FUNCTION_BLOCK PnpCylinders (* Composite Function Block Type *)
  (* Standard: 61499-2 *)
  (* Version 0.0, 2/7/2012, XPMUser, nxtControl GmbH, template *)
  PACKAGE Main;
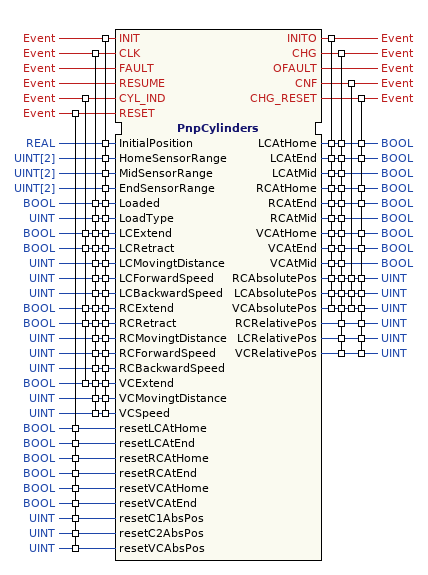
  EVENT_INPUT
    INIT WITH LCForwardSpeed, LCBackwardSpeed, LCExtend, LCRetract, LCMovingtDistance, HomeSensorRange, EndSensorRange, InitialPosition, LoadType, Loaded, MidSensorRange, RCForwardSpeed, RCBackwardSpeed, RCExtend, RCRetract, RCMovingtDistance, VCSpeed, VCExtend, VCMovingtDistance; (* Initialization Request *)
    CLK WITH Loaded, LoadType, LCExtend, LCRetract, LCMovingtDistance, LCForwardSpeed, LCBackwardSpeed, RCExtend, RCRetract, RCMovingtDistance, RCForwardSpeed, RCBackwardSpeed, VCExtend, VCMovingtDistance, VCSpeed;
    FAULT;
    RESUME;
    CYL_IND WITH LCExtend, LCRetract, RCExtend, RCRetract, VCExtend;
    RESET WITH resetLCAtHome, resetLCAtEnd, resetRCAtHome, resetRCAtEnd, resetVCAtHome, resetVCAtEnd, resetC1AbsPos, resetC2AbsPos, resetVCAbsPos;
  END_EVENT
  EVENT_OUTPUT
    INITO WITH LCAtHome, LCAtEnd, LCAtMid, RCAtHome, RCAtEnd, RCAtMid, VCAtHome, VCAtEnd, VCAtMid, RCAbsolutePos, LCAbsolutePos, VCAbsolutePos; (* Initialization Confirm *)
    CHG WITH LCAtHome, LCAtEnd, LCAtMid, RCAtHome, RCAtEnd, RCAtMid, VCAtHome, VCAtEnd, VCAtMid, RCAbsolutePos, LCAbsolutePos, VCAbsolutePos, RCRelativePos, LCRelativePos, VCRelativePos;
    OFAULT;
    CNF WITH RCAbsolutePos, LCAbsolutePos, VCAbsolutePos;
    CHG_RESET WITH LCAtHome, LCAtEnd, RCAtHome, RCAtEnd, VCAtHome, VCAtEnd, RCAbsolutePos, LCAbsolutePos, VCAbsolutePos, RCRelativePos, LCRelativePos, VCRelativePos;
  END_EVENT
  VAR_INPUT
    InitialPosition : REAL; (* Initial position *)
    HomeSensorRange : ARRAY [0..1] OF UINT; (* Detection range of home sensor *)
    MidSensorRange : ARRAY [0..1] OF UINT; (* Detection range of home sensor *)
    EndSensorRange : ARRAY [0..1] OF UINT; (* Detection range of end sensor *)
    Loaded : BOOL;
    LoadType : UINT;
    LCExtend : BOOL;
    LCRetract : BOOL;
    LCMovingtDistance : UINT; (* Moving distance *)
    LCForwardSpeed : UINT; (* Forward speed *)
    LCBackwardSpeed : UINT; (* Backward speed *)
    RCExtend : BOOL;
    RCRetract : BOOL;
    RCMovingtDistance : UINT; (* Moving distance *)
    RCForwardSpeed : UINT; (* Forward speed *)
    RCBackwardSpeed : UINT; (* Backward speed *)
    VCExtend : BOOL;
    VCMovingtDistance : UINT; (* Moving distance *)
    VCSpeed : UINT; (* Forward speed *)
    resetLCAtHome : BOOL;
    resetLCAtEnd : BOOL;
    resetRCAtHome : BOOL;
    resetRCAtEnd : BOOL;
    resetVCAtHome : BOOL;
    resetVCAtEnd : BOOL;
    resetC1AbsPos : UINT;
    resetC2AbsPos : UINT;
    resetVCAbsPos : UINT;
  END_VAR
  VAR_OUTPUT
    LCAtHome : BOOL; (* Detected at home position *)
    LCAtEnd : BOOL; (* Detected at end position *)
    LCAtMid : BOOL;
    RCAtHome : BOOL; (* Detected at home position *)
    RCAtEnd : BOOL; (* Detected at end position *)
    RCAtMid : BOOL;
    VCAtHome : BOOL; (* Detected at home position *)
    VCAtEnd : BOOL; (* Detected at end position *)
    VCAtMid : BOOL;
    RCAbsolutePos : UINT;
    LCAbsolutePos : UINT;
    VCAbsolutePos : UINT;
    RCRelativePos : UINT;
    LCRelativePos : UINT;
    VCRelativePos : UINT;
  END_VAR
  FBS
    LeftCylinder : GenericCylinderModelType1(inputAbsPos := 0);
    RightCylinder : GenericCylinderModelType1(inputAbsPos := 0);
    VerticleCylinder : GenericCylinderModelType2(inputAbsPos := 0);
  END_FBS
  EVENT_CONNECTIONS
    INIT TO LeftCylinder.INIT;
    CLK TO LeftCylinder.CLK;
    FAULT TO LeftCylinder.FAULT;
    RESUME TO LeftCylinder.RESUME;
    VerticleCylinder.INITO TO INITO;
    VerticleCylinder.CHG TO CHG;
    LeftCylinder.OFAULT TO RightCylinder.FAULT;
    RightCylinder.OFAULT TO VerticleCylinder.FAULT;
    VerticleCylinder.OFAULT TO OFAULT;
    RESUME TO RightCylinder.RESUME;
    RESUME TO VerticleCylinder.RESUME;
    VerticleCylinder.CNF TO CNF;
    RightCylinder.CNF TO CNF;
    LeftCylinder.CNF TO CNF;
    LeftCylinder.INITO TO RightCylinder.INIT;
    RightCylinder.INITO TO VerticleCylinder.INIT;
    CYL_IND TO LeftCylinder.CYL_IND;
    CYL_IND TO RightCylinder.CYL_IND;
    CYL_IND TO VerticleCylinder.CYL_IND;
    RESET TO LeftCylinder.RESET;
    LeftCylinder.CHG_RESET TO RightCylinder.RESET;
    RightCylinder.CHG_RESET TO VerticleCylinder.RESET;
    VerticleCylinder.CHG_RESET TO CHG_RESET;
    LeftCylinder.CHG TO RightCylinder.CLK;
    RightCylinder.CHG TO VerticleCylinder.CLK;
  END_CONNECTIONS
  DATA_CONNECTIONS
    LCForwardSpeed TO LeftCylinder.ForwardSpeed;
    LCBackwardSpeed TO LeftCylinder.BackwardSpeed;
    InitialPosition TO LeftCylinder.InitialPosition;
    LCMovingtDistance TO LeftCylinder.MovingtDistance;
    HomeSensorRange TO LeftCylinder.HomeSensorRange;
    MidSensorRange TO LeftCylinder.MidSensorRange;
    EndSensorRange TO LeftCylinder.EndSensorRange;
    LCExtend TO LeftCylinder.Extend;
    LCRetract TO LeftCylinder.Retract;
    Loaded TO LeftCylinder.Loaded;
    LoadType TO LeftCylinder.LoadType;
    RCForwardSpeed TO RightCylinder.ForwardSpeed;
    RCBackwardSpeed TO RightCylinder.BackwardSpeed;
    InitialPosition TO RightCylinder.InitialPosition;
    RCMovingtDistance TO RightCylinder.MovingtDistance;
    HomeSensorRange TO RightCylinder.HomeSensorRange;
    MidSensorRange TO RightCylinder.MidSensorRange;
    EndSensorRange TO RightCylinder.EndSensorRange;
    RCExtend TO RightCylinder.Extend;
    RCRetract TO RightCylinder.Retract;
    Loaded TO RightCylinder.Loaded;
    LoadType TO RightCylinder.LoadType;
    VCSpeed TO VerticleCylinder.ForwardSpeed;
    VCSpeed TO VerticleCylinder.BackwardSpeed;
    InitialPosition TO VerticleCylinder.InitialPosition;
    VCMovingtDistance TO VerticleCylinder.MovingtDistance;
    HomeSensorRange TO VerticleCylinder.HomeSensorRange;
    MidSensorRange TO VerticleCylinder.MidSensorRange;
    EndSensorRange TO VerticleCylinder.EndSensorRange;
    VCExtend TO VerticleCylinder.Extend;
    Loaded TO VerticleCylinder.Loaded;
    LoadType TO VerticleCylinder.LoadType;
    LeftCylinder.AtHome TO LCAtHome;
    LeftCylinder.AtMid TO LCAtMid;
    RightCylinder.AtHome TO RCAtHome;
    RightCylinder.AtMid TO RCAtMid;
    LeftCylinder.AtEnd TO LCAtEnd;
    RightCylinder.AtEnd TO RCAtEnd;
    VerticleCylinder.AtHome TO VCAtHome;
    VerticleCylinder.AtEnd TO VCAtEnd;
    VerticleCylinder.AtMid TO VCAtMid;
    RightCylinder.AbsolutePos TO RCAbsolutePos;
    LeftCylinder.AbsolutePos TO LCAbsolutePos;
    VerticleCylinder.AbsolutePos TO VCAbsolutePos;
    resetLCAtHome TO LeftCylinder.resetAtHome;
    resetLCAtEnd TO LeftCylinder.resetAtEnd;
    resetRCAtHome TO RightCylinder.resetAtHome;
    resetRCAtEnd TO RightCylinder.resetAtEnd;
    resetVCAtHome TO VerticleCylinder.resetAtHome;
    resetVCAtEnd TO VerticleCylinder.resetAtEnd;
    resetC1AbsPos TO LeftCylinder.resetAbsPos;
    resetC2AbsPos TO RightCylinder.resetAbsPos;
    resetVCAbsPos TO VerticleCylinder.resetAbsPos;
    VerticleCylinder.RelativePos TO VCRelativePos;
    RightCylinder.RelativePos TO RCRelativePos;
    LeftCylinder.RelativePos TO LCRelativePos;
  END_CONNECTIONS
END_FUNCTION_BLOCK
